(* IEC 61131-3 sources: Vision2026/PLC_Programs/Mitsubishi_GXWorks3, 6 files *)

(* ---- POU_01_Watchdog_Heartbeat.st ---- *)
(* ========================================================================== *)
(* PROGRAM NAME: POU_01_Watchdog_Heartbeat                                   *)
(* DESCRIPTION : 2-Way Heartbeat Watchdog & Line Safety Interlock (24/7)     *)
(* PLATFORM    : Mitsubishi iQ-R / iQ-F (FX5U) / Q Series (GX Works 3 / 2)   *)
(* ========================================================================== *)

VAR
    fbVisionHeartbeatR_TRIG : R_TRIG;
    fbVisionHeartbeatF_TRIG : F_TRIG;
    bVisionHeartbeatToggled : BOOL;
    tWatchdogTimer : TON;
    tPlcHeartbeatTimer : TON;
END_VAR

(* -------------------------------------------------------------------------- *)
(* 1. TẠO NHỊP TIM PLC ĐẢO 0/1 CHU KỲ 100ms GỬI CHO VISION PC                 *)
(* -------------------------------------------------------------------------- *)
tPlcHeartbeatTimer(IN := NOT tPlcHeartbeatTimer.Q, PT := T#100ms);
IF tPlcHeartbeatTimer.Q THEN
    X0 := NOT X0; (* Đảo bit PLC Heartbeat X0 (hoặc M201) mỗi 100ms *)
END_IF;

(* -------------------------------------------------------------------------- *)
(* 2. GIÁM SÁT NHỊP TIM TỪ VISION PC (Y0 hoặc M200)                            *)
(* Phát hiện cạnh lên (R_TRIG) hoặc cạnh xuống (F_TRIG) của Vision_Heartbeat  *)
(* -------------------------------------------------------------------------- *)
fbVisionHeartbeatR_TRIG(CLK := Y0);
fbVisionHeartbeatF_TRIG(CLK := Y0);
bVisionHeartbeatToggled := fbVisionHeartbeatR_TRIG.Q OR fbVisionHeartbeatF_TRIG.Q;

(* -------------------------------------------------------------------------- *)
(* 3. WATCHDOG TIMER: NẾU QUÁ 300ms KHÔNG THẤY VISION ĐẢO BIT THÌ BÁO LỖI     *)
(* -------------------------------------------------------------------------- *)
tWatchdogTimer(
    IN := NOT bVisionHeartbeatToggled,
    PT := T#300ms
);

IF tWatchdogTimer.Q THEN
    M202 := TRUE;  (* Bật cờ lỗi Vision Fault (Mất kết nối / PC treo) *)
    Y10  := FALSE; (* Ngắt liên động an toàn: Dừng khẩn cấp động cơ chuyền *)
ELSE
    M202 := FALSE; (* Trạng thái truyền thông Vision bình thường *)
    Y10  := TRUE;  (* Cho phép liên động chạy chuyền *)
END_IF;

(* ---- POU_01_Watchdog_Heartbeat_Native.st ---- *)
(* ========================================================================== *)
(* PROGRAM NAME: POU_01_Watchdog_Heartbeat (Native Mitsubishi Version)       *)
(* ĐẶC ĐIỂM    : SIÊU GỌN - KHÔNG CẦN KHAI BÁO LOCAL LABEL PHỨC TẠP          *)
(*               DÙNG TRỰC TIẾP TIMER PHẦN CỨNG T0 VÀ BIT HỆ THỐNG SM410      *)
(* PLATFORM    : Mitsubishi FX5U (GX Works 3)                                *)
(* ========================================================================== *)

(* -------------------------------------------------------------------------- *)
(* 1. TẠO NHỊP TIM PLC ĐẢO 0/1 CHU KỲ 100ms GỬI CHO VISION PC                 *)
(* Sử dụng trực tiếp cờ xung nhịp hệ thống SM410 (100ms clock) của FX5U       *)
(* -------------------------------------------------------------------------- *)
M108 := SM410; (* PLC_Heartbeat xuất liên tục sang Vision PC qua MC Protocol *)

(* -------------------------------------------------------------------------- *)
(* 2. PHÁT HIỆN NHỊP TIM VISION PC (Y0 hoặc M100) ĐẢO TRẠNG THÁI              *)
(* So sánh bit hiện tại với chu kỳ trước: Đảo bit thì kích xung M201 1 vòng   *)
(* -------------------------------------------------------------------------- *)
IF Y0 <> M200 THEN
    M200 := Y0;    (* M200: Bộ đệm lưu trạng thái chu kỳ trước của Y0 *)
    M201 := TRUE;  (* M201: Xung báo Vision PC vừa đảo nhịp tim *)
ELSE
    M201 := FALSE;
END_IF;

(* -------------------------------------------------------------------------- *)
(* 3. WATCHDOG TIMER T0: NẾU QUÁ 300ms KHÔNG THẤY VISION ĐẢO BIT THÌ BÁO LỖI  *)
(* Lệnh OUT_T(điều kiện đếm, tên Timer, giá trị K đặt): K3 = 3 * 100ms = 300ms*)
(* -------------------------------------------------------------------------- *)
OUT_T(NOT M201, T0, 3);

(* -------------------------------------------------------------------------- *)
(* 4. LIÊN ĐỘNG AN TOÀN TOÀN HỆ THỐNG                                         *)
(* -------------------------------------------------------------------------- *)
IF T0 THEN
    M202 := TRUE;  (* Bật cờ lỗi Vision Fault (Mất kết nối hoặc PC treo) *)
    Y10  := FALSE; (* Ngắt liên động an toàn: Dừng khẩn cấp động cơ chuyền *)
ELSE
    M202 := FALSE; (* Truyền thông bình thường *)
    Y10  := TRUE;  (* Cho phép liên động chạy chuyền *)
END_IF;

(* ---- POU_02_Vision_Handshake.st ---- *)
(* ========================================================================== *)
(* PROGRAM NAME: POU_02_Vision_Handshake                                     *)
(* DESCRIPTION : 24/7 Robust Handshake State Machine with Vision System      *)
(* PLATFORM    : Mitsubishi iQ-R / iQ-F (FX5U) / Q Series (GX Works 3 / 2)   *)
(* ========================================================================== *)

VAR
    iState : INT := 0; (* 0: Idle, 10: Triggered, 20: Inspecting, 30: Latched, 40: Ack, 99: Timeout *)
    fbPartSensorR_TRIG : R_TRIG;
    tHandshakeTimeout : TON;
    bPartCapturedOk : BOOL;
    bPartCapturedNg : BOOL;
END_VAR

(* -------------------------------------------------------------------------- *)
(* BẮT CẠNH CẢM BIẾN PHÔI ĐẾN VỊ TRÍ CHỤP (X2)                               *)
(* -------------------------------------------------------------------------- *)
fbPartSensorR_TRIG(CLK := X2);

(* -------------------------------------------------------------------------- *)
(* TIMER BẢO VỆ CHU TRÌNH BẮT TAY (TIMEOUT 2000ms)                            *)
(* -------------------------------------------------------------------------- *)
tHandshakeTimeout(
    IN := (iState > 0 AND iState < 99),
    PT := T#2000ms
);

IF tHandshakeTimeout.Q THEN
    iState := 99; (* Chuyển sang trạng thái xử lý lỗi Timeout *)
END_IF;

(* -------------------------------------------------------------------------- *)
(* MÁY TRẠNG THÁI BẮT TAY CÔNG NGHIỆP 24/7 (STATE MACHINE)                    *)
(* -------------------------------------------------------------------------- *)
CASE iState OF
    0: (* TRẠNG THÁI IDLE: Chờ sản phẩm vào và Vision sẵn sàng *)
        M10 := FALSE; (* Xung trigger OFF *)
        X1  := FALSE; (* Xung Ack OFF *)
        IF fbPartSensorR_TRIG.Q AND Y1 (* Vision_Ready *) AND NOT M202 (* Không có lỗi *) THEN
            M10 := TRUE;   (* Bắn xung Trigger cho Vision PC *)
            iState := 10;
        END_IF;

    10: (* TRẠNG THÁI TRIGGER SENT: Chờ Vision xác nhận nhận lệnh (Vision Busy Y2) *)
        IF Y2 (* Vision_Busy *) THEN
            M10 := FALSE;  (* Ngắt xung Trigger ngay khi Vision đã bận *)
            iState := 20;
        END_IF;

    20: (* TRẠNG THÁI INSPECTING: Chờ Vision phân tích xong (Vision Done Y3) *)
        IF Y3 (* Vision_Done *) THEN
            (* Chốt kết quả kiểm tra *)
            bPartCapturedOk := Y4; (* Vision_Pass *)
            bPartCapturedNg := Y5; (* Vision_NG *)

            (* Nếu sản phẩm NG -> Đẩy vào bộ đệm Shift Register để chờ thổi loại bỏ *)
            IF bPartCapturedNg THEN
                (* Gọi hàm nạp vị trí sản phẩm lỗi vào hàng đợi Reject *)
                M30 := TRUE; (* Kích hoạt cờ nạp Shift Register *)
            END_IF;

            X1 := TRUE; (* Gửi tín hiệu PLC_Ack (X1) xác nhận đã nhận kết quả *)
            iState := 30;
        END_IF;

    30: (* TRẠNG THÁI WAIT VISION RESET: Chờ Vision hạ cờ Done (Y3) *)
        IF NOT Y3 (* Vision_Done hạ về 0 *) THEN
            X1 := FALSE; (* PLC hạ cờ PLC_Ack (X1) hoàn tất chu trình *)
            M30 := FALSE;
            iState := 0; (* Quay về IDLE sẵn sàng cho con hàng tiếp theo *)
        END_IF;

    99: (* TRẠNG THÁI XỬ LÝ LỖI TIMEOUT *)
        M10 := FALSE;
        X1  := FALSE;
        M210 := TRUE; (* Cảnh báo lỗi bắt tay Vision Timeout *)
        (* Tự phục hồi sau khi người dùng bấm Reset M211 hoặc Vision Ready trở lại *)
        IF M211 OR Y1 THEN
            M210 := FALSE;
            M211 := FALSE;
            iState := 0;
        END_IF;
END_CASE;

(* ---- POU_03_Encoder_Tracking.st ---- *)
(* ========================================================================== *)
(* PROGRAM NAME: POU_03_Encoder_Tracking                                     *)
(* DESCRIPTION : High-Speed Counter (HSC) Read, Position mm & Speed Calc     *)
(* PLATFORM    : Mitsubishi iQ-R / iQ-F (FX5U) / Q Series (GX Works 3 / 2)   *)
(* ========================================================================== *)

VAR
    diRawEncoderPulses : DINT;
    diLastEncoderPulses : DINT;
    diDeltaPulses : DINT;
    tSpeedCalcTimer : TON;
    rPulsesPerMm : REAL := 100.0; (* 100 xung = 1 mm di chuyển *)
    rCurrentPositionMm : REAL;
END_VAR

(* -------------------------------------------------------------------------- *)
(* 1. ĐỌC BỘ ĐẾM XUNG TỐC ĐỘ CAO (HIGH SPEED COUNTER)                         *)
(* Đối với FX5U: SD6000 (HSC1 CH1) hoặc C251; Đối với Q-Series: QD62 buffer    *)
(* -------------------------------------------------------------------------- *)
(* Lấy giá trị xung hiện tại từ bộ đếm phần cứng gán vào D1000 (DINT 32-bit)   *)
diRawEncoderPulses := D1000;

(* Tính đổi tọa độ vị trí thực tế của cuộn/băng chuyền theo mm *)
IF rPulsesPerMm > 0.0 THEN
    rCurrentPositionMm := DINT_TO_REAL(diRawEncoderPulses) / rPulsesPerMm;
    (* Lưu tọa độ mm thực tế vào D1004 (REAL 32-bit) *)
    D1004 := rCurrentPositionMm;
END_IF;

(* -------------------------------------------------------------------------- *)
(* 2. TÍNH TỐC ĐỘ DÂY CHUYỀN (m/phút) MỖI CHU KỲ 100ms                        *)
(* -------------------------------------------------------------------------- *)
tSpeedCalcTimer(IN := NOT tSpeedCalcTimer.Q, PT := T#100ms);
IF tSpeedCalcTimer.Q THEN
    diDeltaPulses := diRawEncoderPulses - diLastEncoderPulses;
    diLastEncoderPulses := diRawEncoderPulses;

    (* Tốc độ (m/min) = (Delta Pulses / PulsesPerMm) * (60s / 0.1s) / 1000mm *)
    IF rPulsesPerMm > 0.0 THEN
        D1002 := REAL_TO_INT((DINT_TO_REAL(diDeltaPulses) / rPulsesPerMm) * 0.6);
    END_IF;
END_IF;

(* ---- POU_04_ShiftRegister_Reject.st ---- *)
(* ========================================================================== *)
(* PROGRAM NAME: POU_04_ShiftRegister_Reject                                 *)
(* DESCRIPTION : FIFO Shift Register & Precision Millimeter Reject Piston    *)
(* PLATFORM    : Mitsubishi iQ-R / iQ-F (FX5U) / Q Series (GX Works 3 / 2)   *)
(* ========================================================================== *)

VAR
    aRejectTargets : ARRAY[0..19] OF REAL; (* Bộ đệm lưu tối đa 20 sản phẩm NG đang trôi *)
    iQueueCount : INT := 0;
    fbPushR_TRIG : R_TRIG;
    tRejectPulse : TON;
    bRejectActive : BOOL;
    i : INT;
    j : INT;
    rTargetMm : REAL;
    rCurrentMm : REAL;
    rDistanceSetting : REAL;
    rToleranceSetting : REAL;
END_VAR

(* Đọc các thông số cài đặt *)
rCurrentMm := D1004; (* Tọa độ mm hiện tại *)
rDistanceSetting := INT_TO_REAL(D100); (* Khoảng cách từ Camera đến Trạm Reject, vd 1500 mm *)
rToleranceSetting := INT_TO_REAL(D102); (* Dung sai kích hoạt, vd 10 mm *)
IF rToleranceSetting <= 0.0 THEN
    rToleranceSetting := 10.0;
END_IF;

(* -------------------------------------------------------------------------- *)
(* 1. NẠP SẢN PHẨM LỖI (NG) VÀO HÀNG ĐỢI FIFO KHI NHẬN CỜ M30 TỪ HANDSHAKE   *)
(* -------------------------------------------------------------------------- *)
fbPushR_TRIG(CLK := M30);
IF fbPushR_TRIG.Q THEN
    IF iQueueCount < 20 THEN
        (* Tính vị trí tọa độ mm mà con hàng lỗi này sẽ đến trạm Reject *)
        aRejectTargets[iQueueCount] := rCurrentMm + rDistanceSetting;
        iQueueCount := iQueueCount + 1;
    END_IF;
END_IF;

(* -------------------------------------------------------------------------- *)
(* 2. SO SÁNH VỊ TRÍ THỰC TẾ VÀ KÍCH HOẠT THỔI / GẠT SẢN PHẨM LỖI             *)
(* -------------------------------------------------------------------------- *)
FOR i := 0 TO (iQueueCount - 1) DO
    rTargetMm := aRejectTargets[i];

    (* Kiểm tra nếu phôi đã tiến vào vùng dung sai của trạm Reject *)
    IF (rCurrentMm >= (rTargetMm - rToleranceSetting)) AND
       (rCurrentMm <= (rTargetMm + rToleranceSetting + 50.0)) THEN

        bRejectActive := TRUE; (* Kích hoạt van xylanh / khí nén *)

        (* Dịch chuyển xóa phần tử đã xử lý khỏi hàng đợi FIFO *)
        FOR j := i TO (iQueueCount - 2) DO
            aRejectTargets[j] := aRejectTargets[j + 1];
        END_FOR;
        aRejectTargets[iQueueCount - 1] := 0.0;
        iQueueCount := iQueueCount - 1;
        EXIT;
    END_IF;
END_FOR;

(* -------------------------------------------------------------------------- *)
(* 3. ĐIỀU KHIỂN ĐỘ RỘNG XUNG XYLANH REJECT (100ms)                          *)
(* -------------------------------------------------------------------------- *)
tRejectPulse(IN := bRejectActive, PT := T#100ms);
IF bRejectActive THEN
    Y20 := TRUE; (* Xuất tín hiệu ON cho van xylanh / vòi phun khí Reject *)
    IF tRejectPulse.Q THEN
        Y20 := FALSE;
        bRejectActive := FALSE; (* Ngắt xung hoàn tất 1 lần thổi *)
    END_IF;
ELSE
    Y20 := FALSE;
END_IF;

(* ---- POU_05_Result_Handler.st ---- *)
(* ========================================================================== *)
(* PROGRAM NAME: POU_05_Result_Handler                                       *)
(* DESCRIPTION : Vision Results Processing & Yield Counters (DINT 32-bit)    *)
(* PLATFORM    : Mitsubishi iQ-R / iQ-F (FX5U) / Q Series (GX Works 3 / 2)   *)
(* ========================================================================== *)

VAR
    fbPassR_TRIG : R_TRIG;
    fbNgR_TRIG : R_TRIG;
    rCurrentOriginX : REAL;
    rCurrentOriginY : REAL;
    rCurrentOriginAngle : REAL;
    rCurrentDistance1 : REAL;
END_VAR

(* -------------------------------------------------------------------------- *)
(* 1. ĐỌC DỮ LIỆU ĐO ĐẠC VÀ TỌA ĐỘ TRUYỀN TỪ VISION VÀO THANH GHI PLC         *)
(* Vision gửi giá trị vào D200 (X), D202 (Y), D204 (Angle), D210 (Distance1)  *)
(* -------------------------------------------------------------------------- *)
rCurrentOriginX     := D200;
rCurrentOriginY     := D202;
rCurrentOriginAngle := D204;
rCurrentDistance1   := D210;

(* -------------------------------------------------------------------------- *)
(* 2. CỘNG DỒN BỘ ĐẾM SỐ LƯỢNG SẢN PHẨM KIỂM TRA (TOTAL, OK, NG)             *)
(* -------------------------------------------------------------------------- *)
fbPassR_TRIG(CLK := Y4); (* Cạnh lên của Vision_Pass *)
fbNgR_TRIG(CLK := Y5);   (* Cạnh lên của Vision_NG *)

IF fbPassR_TRIG.Q THEN
    D300 := D300 + 1; (* Tăng tổng số kiểm tra D300 *)
    D302 := D302 + 1; (* Tăng tổng số OK D302 *)
END_IF;

IF fbNgR_TRIG.Q THEN
    D300 := D300 + 1; (* Tăng tổng số kiểm tra D300 *)
    D304 := D304 + 1; (* Tăng tổng số NG D304 *)
END_IF;

(* -------------------------------------------------------------------------- *)
(* 3. NÚT NHẤN RESET BỘ ĐẾM SẢN LƯỢNG (HMI / NÚT NHẤN M310)                  *)
(* -------------------------------------------------------------------------- *)
IF M310 THEN
    D300 := 0;
    D302 := 0;
    D304 := 0;
    M310 := FALSE;
END_IF;
